// TIA Portal V19 export
FUNCTION_BLOCK "TYPIC_C104_IF_LBS"   // FB93, FBD
TITLE = TYPIC_C104_IF_LBS: Luchtbehandelingssysteem
{ S7_Optimized_Access := 'TRUE' }
AUTHOR : OCOTECH
FAMILY : Typical
NAME : C104.704
// Logisch Object Besturing: C104.704
// 
// De interne functie Luchtbehandelingssysteem verzorgt de bewaking van het luchtbehandelingssysteem van een noodstroomaggregaat.
// stored: MemoryReserve 10, SetENOAutomatically false
   VAR_INPUT
      EXT_AUT { ExternalAccessible := 'False'; ExternalVisible := 'False'; ExternalWritable := 'False'} : Bool;   // Externe (hoofd) beveiliging (1 = OK)
      EXT_HW { ExternalAccessible := 'False'; ExternalVisible := 'False'; ExternalWritable := 'False'} : Bool;   // Sturings hardware (PLC) bewaking (1 = OK)
      IN_STO_NOK { ExternalAccessible := 'False'; ExternalVisible := 'False'; ExternalWritable := 'False'} : Bool;   // Storing aanwezig die niet observeerbaar tot gevolg heeft
      IN_STO_OK { ExternalAccessible := 'False'; ExternalVisible := 'False'; ExternalWritable := 'False'} : Bool;   // Storing aanwezig die observeerbaarheid niet beinvloed
      IN_KLP_OPEN { ExternalAccessible := 'False'; ExternalVisible := 'False'; ExternalWritable := 'False'} : Bool;   // Kleppenregister open
      IN_KLP_TOE { ExternalAccessible := 'False'; ExternalVisible := 'False'; ExternalWritable := 'False'} : Bool;   // Kleppenregister dicht
      IN_VEN_AAN { ExternalAccessible := 'False'; ExternalVisible := 'False'; ExternalWritable := 'False'} : Bool;   // Ventilator aan
      IN_AUT_C104 { ExternalAccessible := 'False'; ExternalVisible := 'False'; ExternalWritable := 'False'} : Bool;   // Beveiligingen: serie geschakelde terugmelding (1 = OK)
   END_VAR
   VAR_OUTPUT
      VAR_IF_OPT { ExternalAccessible := 'False'; ExternalVisible := 'False'; ExternalWritable := 'False'} : "C104_VAR_IF_OPT_TYPIC";   // Struct met alle variabelen naar bovenliggende functies
   END_VAR
   VAR
      STO { ExternalWritable := 'False'} : Struct   // Storingen
         A001 : Bool;   // Beveiliging aangesproken
         A002 : Bool;   // Luchtbehandelingssysteem in storing
         A003 : Bool;   // Algemene storing luchtbehandelingssysteem
      END_STRUCT;
      VAR { ExternalWritable := 'False'} : Struct   // Variabelen
         KLP_OPEN { ExternalAccessible := 'False'; ExternalVisible := 'False'} : Bool;   // Kleppenregister open
         KLP_TOE { ExternalAccessible := 'False'; ExternalVisible := 'False'} : Bool;   // Kleppenregister dicht
         VEN_AAN { ExternalAccessible := 'False'; ExternalVisible := 'False'} : Bool;   // Ventilator aan
         EXT_AUT { ExternalAccessible := 'False'; ExternalVisible := 'False'} : Bool;   // Externe (hoofd) beveiliging aangesproken
         EXT_HW { ExternalAccessible := 'False'; ExternalVisible := 'False'} : Bool;   // Sturings hardware (PLC) in storing
      END_STRUCT;
   END_VAR
BEGIN

REGION Network 1: START
END_REGION

REGION Network 2: +++ Verwerking statussen +++
   // Bepalen van de statussen van het luchtbehandelingssysteem.
END_REGION

REGION Network 3: +++ Storingen +++
   // Verwerken van de storingsmeldingen (inputs).
END_REGION

REGION Network 4: Storing A001: Beveiliging aangesproken
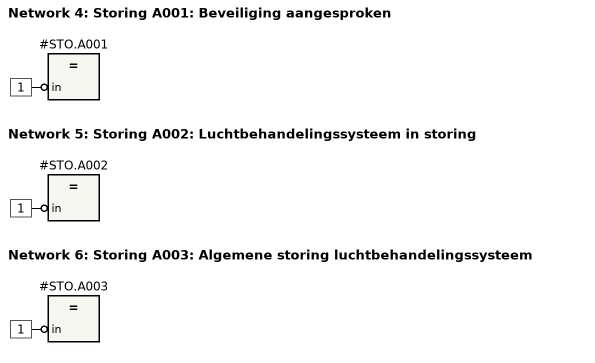
   #STO.A001 := NOT 1;
END_REGION

REGION Network 5: Storing A002: Luchtbehandelingssysteem in storing
   #STO.A002 := NOT 1;
END_REGION

REGION Network 6: Storing A003: Algemene storing luchtbehandelingssysteem
   #STO.A003 := NOT 1;
END_REGION

REGION Network 7 (SCL): EINDE
   // Variabelen van intern scada rakvlak naar outputs copieren
   #VAR_IF_OPT.KLP_OPEN := #VAR.KLP_OPEN;
   #VAR_IF_OPT.KLP_TOE := #VAR.KLP_TOE;
   #VAR_IF_OPT.VEN_AAN := #VAR.VEN_AAN;
   #VAR_IF_OPT.EXT_AUT := #VAR.EXT_AUT;
   #VAR_IF_OPT.EXT_HW := #VAR.EXT_HW;
   #VAR_IF_OPT.STO := #STO;
END_REGION
END_FUNCTION_BLOCK
